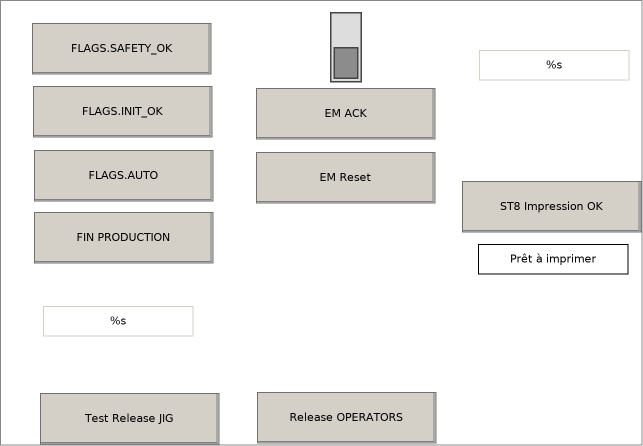
VISUALIZATION Visualization  // 643x446
    Button (32,23 179x51), "FLAGS.SAFETY_OK"
        toggle Flag_Variables.FLAGS.SAFETY_OK
    Button (33,86 179x51), "FLAGS.INIT_OK"
        toggle Flag_Variables.FLAGS.INIT_OK
    Button (34,150 179x51), "FLAGS.AUTO"
        toggle Flag_Variables.FLAGS.AUTO
    Button (256,88 179x51), "EM ACK"
        tap Flag_Variables.SAFETY_OUT.NOT_AUS_ErrAck
    Button (256,152 179x51), "EM Reset"
        tap Flag_Variables.SAFETY_OUT.NOT_AUS_RESET
    DipSwitch (311,12 70x70), variable: Flag_Variables.SAFETY_OUT.NOT_AUS_RUN, behaviour: TOGGLE, style: Switch-DipSwitch-Gray
    Textfield (479,50 150x30), "%s", text variable: Flag_Variables.SAFETY_IN.NOT_AUS_State
    Textfield (43,306 150x30), "%s", text variable: GEMMA.STEP
    Button (34,212 179x51), "FIN PRODUCTION"
        tap GEMMA.F2_END
    Button (40,393 179x51), "Test Release JIG"
        tap CONVEYOR.TEST_RELEASE
    Button (257,392 179x51), "Release OPERATORS"
        tap Flag_Variables.FLAGS.DEBUG_OPERATOR
    Button (462,181 179x51), "ST8 Impression OK"
        tap IOs_Variables.ST8_IMPRESSION_OK
    Rectangle (478,244 150x30), "Prêt à imprimer", colour toggle: IOs_Variables.ST8_PRET_A_IMPRIMER
END_VISUALIZATION

(* stored: Version 1.1.0.1, ProductVersion 3.1.0.26
   Visu Visualization: Id {813f2506-94fd-469a-9988-98ea7a6fd1cb} *)
